{attribute 'GeneratedUsingTerminal: EP9521-0020-0000'}
{attribute addProperty BoxType "EP9521-0020-0000"}
{attribute addProperty Id "A_0025_EP9576_1032_0016EP9576_F397F1AC21"}
{attribute addProperty CRC "4039103825"}
{attribute addProperty Size "21"}
TYPE A_0024_EP9521_0020_0000_F0BFD551 EXTENDS EP9521_1FC0878B :
STRUCT
	{attribute addProperty Name "A_0025_EP9576_1032_0016"}
	{attribute addProperty PreviousPort "A_0024(EP9521-0020-0000) : B"}
	A_0025_EP9576_1032_0016 : EP9576_F397F1AC;
END_STRUCT
END_TYPE

(* stored: Version 1.2.0.0, ProductVersion 3.1.4024.9
   DUT A_0024_EP9521_0020_0000_F0BFD551: Id {854cffe6-b4da-4a04-b029-9d621db0277a} *)
